// TwinCAT 3 PLC project MotorRuntime
// ProgramVersion: 3.1.4026.24
// libraries:
//   Tc2_Standard, * (Beckhoff Automation GmbH)
//   Tc2_System, * (Beckhoff Automation GmbH)
//   Tc3_Module, * (Beckhoff Automation GmbH)
// project tree:
//   DUTs/ DUT_AllocationSample.TcDUT, DUT_AxisCalibration.TcDUT, DUT_CommutationOverride.TcDUT, DUT_MotorDriverCommand.TcDUT, DUT_MotorDriverStatus.TcDUT, DUT_MotorFeedbackSnapshot.TcDUT
//   GVLs/ GVL_AllocationTransfer.TcGVL, GVL_MotorRuntime.TcGVL, GVL_MotorRuntimeInternal.TcGVL
//   POUs/ FB_AllocationTransfer.TcPOU, F_ArchRadToCstcaAngle.TcPOU, F_ArchWrap2Pi.TcPOU, FB_MotorCommandArbiter.TcPOU, FB_MotorIoWatchdog.TcPOU, FB_MotorRuntimeKernel.TcPOU, PRG_MotorRuntime.TcPOU
//   / PlcTask.TcTTO
// (motion and I/O tree: see PLC project experimentsequencer)
// real-time tasks:
//   TASK PlcTask1: cycle T#250us, priority 21, ADS port 351
//   TASK PlcTask: cycle T#125us, priority 20, ADS port 350
//   TASK StateTask: cycle T#10ms, priority 1, ADS port 352
// variable links:
//   ExperimentSequencer/ExperimentSequencer Instance <-> MotorRuntime/MotorRuntime Instance
//     PlcTask Inputs/GVL_ExperimentSequencer.motorFeedback <-> PlcTask Outputs/GVL_MotorRuntimeInternal.Feedback
//     PlcTask Outputs/GVL_ExperimentSequencer.commutationOverride <-> PlcTask Inputs/GVL_MotorRuntimeInternal.CommutationOverride
//     PlcTask Outputs/GVL_ExperimentSequencer.driveCommand <-> PlcTask Inputs/GVL_MotorRuntimeInternal.CommissioningCommand
//   MotorRuntime/MotorRuntime Instance <-> Device 3 (EtherCAT)/Drive 7 (XE2)
//     PlcTask Inputs/PRG_MotorRuntime.copleyActualCurrentCountModule1 <-> Module 1 (Cyclic torque with commutation angle Mode)/Cyclic torque with commutation angle Inputs/Torque actual value
//     PlcTask Inputs/PRG_MotorRuntime.copleyActualCurrentCountModule2 <-> Module 2 (Cyclic torque with commutation angle Mode)/Cyclic torque with commutation angle Inputs/Torque actual value
//     PlcTask Inputs/PRG_MotorRuntime.copleyInputToggle <-> WcState/InputToggle
//     PlcTask Inputs/PRG_MotorRuntime.copleyStatusWordModule1 <-> Module 1 (Cyclic torque with commutation angle Mode)/Cyclic torque with commutation angle Inputs/Status word
//     PlcTask Inputs/PRG_MotorRuntime.copleyStatusWordModule2 <-> Module 2 (Cyclic torque with commutation angle Mode)/Cyclic torque with commutation angle Inputs/Status word
//     PlcTask Inputs/PRG_MotorRuntime.copleyWcState <-> WcState/WcState
//     PlcTask Outputs/PRG_MotorRuntime.copleyCommutationAngleModule1 <-> Module 1 (Cyclic torque with commutation angle Mode)/Cyclic torque with commutation angle Outputs/Commutation angle
//     PlcTask Outputs/PRG_MotorRuntime.copleyCommutationAngleModule2 <-> Module 2 (Cyclic torque with commutation angle Mode)/Cyclic torque with commutation angle Outputs/Commutation angle
//     PlcTask Outputs/PRG_MotorRuntime.copleyControlWordModule1 <-> Module 1 (Cyclic torque with commutation angle Mode)/Cyclic torque with commutation angle Outputs/Control word
//     PlcTask Outputs/PRG_MotorRuntime.copleyControlWordModule2 <-> Module 2 (Cyclic torque with commutation angle Mode)/Cyclic torque with commutation angle Outputs/Control word
//     PlcTask Outputs/PRG_MotorRuntime.copleyTargetTorqueModule1 <-> Module 1 (Cyclic torque with commutation angle Mode)/Cyclic torque with commutation angle Outputs/Target Torque
//     PlcTask Outputs/PRG_MotorRuntime.copleyTargetTorqueModule2 <-> Module 2 (Cyclic torque with commutation angle Mode)/Cyclic torque with commutation angle Outputs/Target Torque
//   MotorRuntime/MotorRuntime Instance <-> Device 3 (EtherCAT)/Drive 8 (XE2)
//     PlcTask Inputs/PRG_MotorRuntime.copleyActualCurrentCountModule3 <-> Module 1 (Cyclic torque with commutation angle Mode)/Cyclic torque with commutation angle Inputs/Torque actual value
//     PlcTask Inputs/PRG_MotorRuntime.copleyActualCurrentCountModule4 <-> Module 2 (Cyclic torque with commutation angle Mode)/Cyclic torque with commutation angle Inputs/Torque actual value
//     PlcTask Inputs/PRG_MotorRuntime.copleyInputToggleDrive2 <-> WcState/InputToggle
//     PlcTask Inputs/PRG_MotorRuntime.copleyStatusWordModule3 <-> Module 1 (Cyclic torque with commutation angle Mode)/Cyclic torque with commutation angle Inputs/Status word
//     PlcTask Inputs/PRG_MotorRuntime.copleyStatusWordModule4 <-> Module 2 (Cyclic torque with commutation angle Mode)/Cyclic torque with commutation angle Inputs/Status word
//     PlcTask Inputs/PRG_MotorRuntime.copleyWcStateDrive2 <-> WcState/WcState
//     PlcTask Outputs/PRG_MotorRuntime.copleyCommutationAngleModule3 <-> Module 1 (Cyclic torque with commutation angle Mode)/Cyclic torque with commutation angle Outputs/Commutation angle
//     PlcTask Outputs/PRG_MotorRuntime.copleyCommutationAngleModule4 <-> Module 2 (Cyclic torque with commutation angle Mode)/Cyclic torque with commutation angle Outputs/Commutation angle
//     PlcTask Outputs/PRG_MotorRuntime.copleyControlWordModule3 <-> Module 1 (Cyclic torque with commutation angle Mode)/Cyclic torque with commutation angle Outputs/Control word
//     PlcTask Outputs/PRG_MotorRuntime.copleyControlWordModule4 <-> Module 2 (Cyclic torque with commutation angle Mode)/Cyclic torque with commutation angle Outputs/Control word
//     PlcTask Outputs/PRG_MotorRuntime.copleyTargetTorqueModule3 <-> Module 1 (Cyclic torque with commutation angle Mode)/Cyclic torque with commutation angle Outputs/Target Torque
//     PlcTask Outputs/PRG_MotorRuntime.copleyTargetTorqueModule4 <-> Module 2 (Cyclic torque with commutation angle Mode)/Cyclic torque with commutation angle Outputs/Target Torque
//   MotorRuntime/MotorRuntime Instance <-> Device 3 (EtherCAT)/Term 1 (EK1100)/Term 2 (EL5042)
//     PlcTask Inputs/PRG_MotorRuntime.encoderError <-> FB Inputs Channel 1/Status/Error
//     PlcTask Inputs/PRG_MotorRuntime.encoderInputToggle <-> WcState/InputToggle
//     PlcTask Inputs/PRG_MotorRuntime.encoderPositionRaw <-> FB Inputs Channel 1/Position
//     PlcTask Inputs/PRG_MotorRuntime.encoderReady <-> FB Inputs Channel 1/Status/Ready
//     PlcTask Inputs/PRG_MotorRuntime.encoderTxPdoState <-> FB Inputs Channel 1/Status/TxPDO State
//     PlcTask Inputs/PRG_MotorRuntime.encoderWcState <-> WcState/WcState
//   MotorRuntime/MotorRuntime Instance <-> TcCOM Objects/Object1 (motor_config)
//     PlcTask Inputs/GVL_MotorRuntime.Command/ControlWord <-> motor_config_Y/controlWord
//     PlcTask Outputs/GVL_MotorRuntime.Status/StatusWord <-> motor_config_U/statusWord
//   MotorRuntime/MotorRuntime Instance <-> TcCOM Objects/Object3 (linear_exp_2025a)
//     PlcTask Inputs/GVL_MotorRuntime.Command/TargetTorque <-> TcModuleOutput/LinearSystem/TargetTorque
//     PlcTask Outputs/GVL_MotorRuntime.Status/PositionActualValue <-> TcModuleInput/LinearSystem/Positionactualvalue
//     PlcTask Outputs/GVL_MotorRuntime.Status/TorqueActualValue <-> TcModuleInput/LinearSystem/Torqueactualvalue1
//     PlcTask Outputs/GVL_MotorRuntime.Status/VelocityActualValue <-> TcModuleInput/LinearSystem/Velocityactualvalue
//   MotorRuntime/MotorRuntime Instance <-> TcCOM Objects/Object3 (linear_exp_tunable_2025a)
//     PlcTask Inputs/GVL_MotorRuntime.Command/TargetTorque <-> TcModuleOutput/linearsystem/TargetTorque
//     PlcTask Outputs/GVL_MotorRuntime.Status/PositionActualValue <-> TcModuleInput/linearsystem/PositionActualValue
//     PlcTask Outputs/GVL_MotorRuntime.Status/TorqueActualValue <-> TcModuleInput/linearsystem/TorqueActualValue
//     PlcTask Outputs/GVL_MotorRuntime.Status/VelocityActualValue <-> TcModuleInput/linearsystem/VelocityActualValue

CONFIGURATION MotorRuntime
    RESOURCE PLC ON TwinCAT3
        TASK PlcTask(INTERVAL := T#250us, PRIORITY := 21);
        PROGRAM PRG_MotorRuntime WITH PlcTask : PRG_MotorRuntime;
    END_RESOURCE
END_CONFIGURATION

// ---- DUTs/DUT_AllocationSample.TcDUT
TYPE DUT_AllocationSample : STRUCT
    cycleIndex : UDINT;
    positionCount : DINT;
    velocityCount : DINT;
    virtualTorque : DINT;
    targetCurrent : ARRAY [1..4] OF DINT;
    actualCurrent : ARRAY [1..4] OF DINT;
    statusWord : ARRAY [1..4] OF DINT;
    faultId : UDINT;
    ioReady : DINT;
    period100ns : UDINT;
    requestId : UDINT;
END_STRUCT
END_TYPE

// ---- DUTs/DUT_AxisCalibration.TcDUT
TYPE DUT_AxisCalibration : STRUCT
    reference_position_count      : DINT;
    reference_commutation_angle   : UINT;
    electrical_direction          : INT;
END_STRUCT
END_TYPE

// ---- DUTs/DUT_CommutationOverride.TcDUT
TYPE DUT_CommutationOverride : STRUCT
    enable                 : BOOL;
    angle_offset_rad       : LREAL;
    axis_index             : UINT;
END_STRUCT
END_TYPE

// ---- DUTs/DUT_MotorDriverCommand.TcDUT
TYPE DUT_MotorDriverCommand : STRUCT
    ControlWord  : WORD;
    TargetTorque : INT;
END_STRUCT
END_TYPE

// ---- DUTs/DUT_MotorDriverStatus.TcDUT
TYPE DUT_MotorDriverStatus : STRUCT
    StatusWord          : WORD;
    PositionActualValue : DINT;
    VelocityActualValue : DINT;
    TorqueActualValue   : INT;
END_STRUCT
END_TYPE

// ---- DUTs/DUT_MotorFeedbackSnapshot.TcDUT
TYPE DUT_MotorFeedbackSnapshot : STRUCT
    encoder_position_raw       : DINT;
    encoder_velocity_raw       : DINT;
    copley_statusword          : WORD;
    copley_actual_current_count: INT;
    output_torque_count        : INT;
    fault_id                   : UDINT;
END_STRUCT
END_TYPE

// ---- GVLs/GVL_AllocationTransfer.TcGVL
{attribute 'qualified_only'}
VAR_GLOBAL CONSTANT
    SCHEMA_VERSION : UDINT := 2;
    SAMPLE_BYTES : UDINT := 80;
END_VAR
VAR_GLOBAL
    // Write parameters first, RequestId last. They are latched only at idle.
    RequestId : UDINT;
    RequestedEnabled : BOOL;
    RequestedPair : UINT := 1;
    RequestedBeta : LREAL;
    RequestedRatio : LREAL := 1.0;
    AckId : UDINT;
    RejectId : UDINT;
    Active : BOOL;
    Started : BOOL;
    Complete : BOOL;
    Pair : UINT;
    Beta : LREAL;
    Ratio : LREAL;
    Weights : ARRAY [1..2] OF LREAL := [1.0,1.0];
    FaultId : UDINT;
    // One coherent cycle is recorded by the common Simulink File Writer.
    Snapshot AT %Q* : DUT_AllocationSample;
END_VAR

// ---- GVLs/GVL_MotorRuntime.TcGVL
{attribute 'qualified_only'}
VAR_GLOBAL
    // The complete public virtual-CST boundary.
    Command AT %I* : DUT_MotorDriverCommand;
    Status  AT %Q* : DUT_MotorDriverStatus;
END_VAR

// ---- GVLs/GVL_MotorRuntimeInternal.TcGVL
{attribute 'qualified_only'}
VAR_GLOBAL CONSTANT
    AXIS_COUNT                    : UINT := 4;
    // Compile-time normal-CST topology: FALSE drives axes 1+2; TRUE drives axes 1..4.
    NORMAL_FOUR_AXIS_ENABLED      : BOOL := TRUE;
    COUNTS_PER_ELECTRICAL_PERIOD : DINT := 360000;
    // Public virtual CST follows CiA 402 rated torque / 1000. The physical
    // Copley channels retain their high-resolution 0.1 A / 1000 scaling.
    VIRTUAL_RATED_TORQUE_EQUIVALENT_CURRENT_MA : DINT := 2000;
    COPLEY_INTERNAL_CURRENT_MA_PER_1000_COUNT   : DINT := 100;
    // Inclusive raw Panasonic encoder windows. Adjacent windows overlap over
    // the measured Core1~2, Core2~3, and Core3~4 transition regions.
    TORQUE_LINKAGE_LOWER_COUNT : ARRAY [1..AXIS_COUNT] OF DINT := [
        54054804, 55809159, 59369714, 63068811];
    TORQUE_LINKAGE_UPPER_COUNT : ARRAY [1..AXIS_COUNT] OF DINT := [
        57600015, 61230980, 64809681, 66655810];
    // Each boundary may vary by 10% of the largest measured segment width:
    // ceil((61230980 - 59369714) * 0.10). Extend both ends for either direction.
    TORQUE_LINKAGE_MARGIN_COUNT : DINT := 186127;
END_VAR

VAR_GLOBAL RETAIN
    // Registered values for all four axes mirror the checked-in authoritative
    // manifest. Set validity false before replacing any complete record.
    RegisteredReferenceValid : ARRAY [1..AXIS_COUNT] OF BOOL := [TRUE, TRUE, TRUE, TRUE];
    RegisteredReference : ARRAY [1..AXIS_COUNT] OF DUT_AxisCalibration := [
        (reference_position_count := 54984708,
         reference_commutation_angle := 49480,
         electrical_direction := 1),
        (reference_position_count := 58408617,
         reference_commutation_angle := 17933,
         electrical_direction := 1),
        (reference_position_count := 61902867,
         reference_commutation_angle := 63448,
         electrical_direction := 1),
        (reference_position_count := 65824016,
         reference_commutation_angle := 57717,
         electrical_direction := 1)
    ];
END_VAR

VAR_GLOBAL
    // Commissioning writes provisional/interim references here. Normal CST
    // never reads this non-retained array.
    CommissioningReference : ARRAY [1..AXIS_COUNT] OF DUT_AxisCalibration;

    // These linked process-image symbols are private commissioning channels.
    // They are deliberately excluded from GVL_MotorRuntime.
    CommissioningCommand AT %I* : DUT_MotorDriverCommand;
    CommutationOverride  AT %I* : DUT_CommutationOverride;

    // One-shot operator acknowledgement for a latched I/O-watchdog fault.
    // PRG_MotorRuntime clears this after sampling it. A reset is accepted only
    // while the selected command is explicitly zero and both slaves are healthy.
    IoWatchdogResetRequest : BOOL;

    // Private commissioning feedback.
    Feedback AT %Q* : DUT_MotorFeedbackSnapshot;
END_VAR

// ---- POUs/PRG_MotorRuntime.TcPOU
PROGRAM PRG_MotorRuntime
VAR
    fbMotor : FB_MotorRuntimeKernel;
    fbArbiter : FB_MotorCommandArbiter;
    fbIoWatchdog : FB_MotorIoWatchdog;
    fbAllocation : FB_AllocationTransfer;

    AllocationRequestId AT %I* : UDINT;

    encoderPositionRaw        AT %I* : ULINT;
    encoderReady              AT %I* : BOOL;
    encoderError              AT %I* : BOOL;
    encoderTxPdoState         AT %I* : BOOL;
    encoderWcState            AT %I* : BOOL;
    encoderInputToggle        AT %I* : BOOL;
    copleyWcState             AT %I* : BOOL;
    copleyInputToggle         AT %I* : BOOL;
    copleyWcStateDrive2       AT %I* : BOOL;
    copleyInputToggleDrive2   AT %I* : BOOL;
    copleyStatusWordModule1         AT %I* : WORD;
    copleyActualCurrentCountModule1 AT %I* : INT;
    copleyStatusWordModule2         AT %I* : WORD;
    copleyActualCurrentCountModule2 AT %I* : INT;
    copleyStatusWordModule3         AT %I* : WORD;
    copleyActualCurrentCountModule3 AT %I* : INT;
    copleyStatusWordModule4         AT %I* : WORD;
    copleyActualCurrentCountModule4 AT %I* : INT;

    copleyControlWordModule1      AT %Q* : WORD;
    copleyTargetTorqueModule1     AT %Q* : INT;
    copleyCommutationAngleModule1 AT %Q* : UINT;
    copleyControlWordModule2      AT %Q* : WORD;
    copleyTargetTorqueModule2     AT %Q* : INT;
    copleyCommutationAngleModule2 AT %Q* : UINT;
    copleyControlWordModule3      AT %Q* : WORD;
    copleyTargetTorqueModule3     AT %Q* : INT;
    copleyCommutationAngleModule3 AT %Q* : UINT;
    copleyControlWordModule4      AT %Q* : WORD;
    copleyTargetTorqueModule4     AT %Q* : INT;
    copleyCommutationAngleModule4 AT %Q* : UINT;

    copleyStatusWord         : ARRAY [1..GVL_MotorRuntimeInternal.AXIS_COUNT] OF WORD;
    copleyActualCurrentCount : ARRAY [1..GVL_MotorRuntimeInternal.AXIS_COUNT] OF INT;
    encoderPositionActualRaw : DINT;
    encoderVelocityActualRaw : DINT;
    previousEncoderPositionRaw : DINT;
    encoderPositionInitialized : BOOL;
    taskIndex                  : DINT;
    cycleTime100ns             : UDINT;
    taskPeriod_s               : LREAL := 0.00025;
END_VAR

taskIndex := GETCURTASKINDEXEX();
IF taskIndex > 0 THEN
    cycleTime100ns := TwinCAT_SystemInfoVarList._TaskInfo[taskIndex].CycleTime;
    IF cycleTime100ns > 0 THEN
        taskPeriod_s := UDINT_TO_LREAL(cycleTime100ns) * 1.0E-7;
    END_IF
END_IF

encoderPositionActualRaw := ULINT_TO_DINT(encoderPositionRaw);
IF encoderPositionInitialized THEN
    // Position is 0.1 um/count; velocity is published in 1 um/s/count.
    encoderVelocityActualRaw := LREAL_TO_DINT(
        DINT_TO_LREAL(encoderPositionActualRaw - previousEncoderPositionRaw)
        * 0.1 / taskPeriod_s);
ELSE
    encoderVelocityActualRaw := 0;
    encoderPositionInitialized := TRUE;
END_IF
previousEncoderPositionRaw := encoderPositionActualRaw;

copleyStatusWord[1] := copleyStatusWordModule1;
copleyActualCurrentCount[1] := copleyActualCurrentCountModule1;
copleyStatusWord[2] := copleyStatusWordModule2;
copleyActualCurrentCount[2] := copleyActualCurrentCountModule2;
copleyStatusWord[3] := copleyStatusWordModule3;
copleyActualCurrentCount[3] := copleyActualCurrentCountModule3;
copleyStatusWord[4] := copleyStatusWordModule4;
copleyActualCurrentCount[4] := copleyActualCurrentCountModule4;

fbArbiter(
    NormalCommand := GVL_MotorRuntime.Command,
    CommissioningCommand := GVL_MotorRuntimeInternal.CommissioningCommand,
    CommutationOverride := GVL_MotorRuntimeInternal.CommutationOverride);

fbMotor(
    Command := fbArbiter.SelectedCommand,
    CommutationOverride := fbArbiter.SelectedCommutationOverride,
    RegisteredReferenceValid := GVL_MotorRuntimeInternal.RegisteredReferenceValid,
    RegisteredReference := GVL_MotorRuntimeInternal.RegisteredReference,
    CommissioningReference := GVL_MotorRuntimeInternal.CommissioningReference,
    EncoderPositionActualRaw := encoderPositionActualRaw,
    EncoderVelocityActualRaw := encoderVelocityActualRaw,
    CopleyStatusWord := copleyStatusWord,
    CopleyActualCurrentCount := copleyActualCurrentCount);

fbIoWatchdog(
    TaskPeriod_s := taskPeriod_s,
    EncoderWcState := encoderWcState,
    EncoderInputToggle := encoderInputToggle,
    EncoderReady := encoderReady,
    EncoderError := encoderError,
    EncoderTxPdoState := encoderTxPdoState,
    CopleyWcState := copleyWcState,
    CopleyInputToggle := copleyInputToggle,
    Copley2WcState := copleyWcStateDrive2,
    Copley2InputToggle := copleyInputToggleDrive2,
    ResetRequest :=
        GVL_MotorRuntimeInternal.IoWatchdogResetRequest
        AND (fbArbiter.CommissioningActive
             OR NOT fbArbiter.CommissioningActive),
    CommandIsZero :=
        (fbArbiter.SelectedCommand.ControlWord = WORD#16#0000)
        AND (fbArbiter.SelectedCommand.TargetTorque = 0));
// Consume the operator acknowledgement as a one-cycle request. Keeping it
// separate from the command prevents automatic re-arm after communication
// recovers while an idle 0/0 command happens to be present.
GVL_MotorRuntimeInternal.IoWatchdogResetRequest := FALSE;

fbAllocation(
    Command := fbArbiter.SelectedCommand,
    RuntimeRequestId := AllocationRequestId,
    CommissioningActive := fbArbiter.CommissioningActive,
    SourceControl := fbMotor.CopleyControlWord,
    SourceTorque := fbMotor.CopleyTargetTorque,
    StatusWord := copleyStatusWord,
    ActualCurrent := copleyActualCurrentCount,
    PositionCount := encoderPositionActualRaw,
    VelocityCount := encoderVelocityActualRaw,
    IoReady := fbIoWatchdog.SafeToDrive,
    SourceFaultId := fbMotor.FaultId,
    Period100ns := cycleTime100ns);

GVL_MotorRuntime.Status := fbMotor.Status;
GVL_MotorRuntimeInternal.Feedback := fbMotor.Feedback;
IF GVL_AllocationTransfer.FaultId <> 0 THEN
    GVL_MotorRuntimeInternal.Feedback.fault_id := GVL_AllocationTransfer.FaultId;
END_IF
IF (fbArbiter.CommissioningActive OR NOT fbArbiter.CommissioningActive)
   AND fbIoWatchdog.Fault THEN
    GVL_MotorRuntimeInternal.Feedback.fault_id := fbIoWatchdog.FaultId;
END_IF

IF (fbArbiter.CommissioningActive OR NOT fbArbiter.CommissioningActive)
   AND fbIoWatchdog.SafeToDrive THEN
    copleyControlWordModule1 := fbAllocation.Control[1];
    copleyTargetTorqueModule1 := fbAllocation.Torque[1];
    copleyCommutationAngleModule1 := fbMotor.CopleyCommutationAngle[1];
    copleyControlWordModule2 := fbAllocation.Control[2];
    copleyTargetTorqueModule2 := fbAllocation.Torque[2];
    copleyCommutationAngleModule2 := fbMotor.CopleyCommutationAngle[2];
    copleyControlWordModule3 := fbAllocation.Control[3];
    copleyTargetTorqueModule3 := fbAllocation.Torque[3];
    copleyCommutationAngleModule3 := fbMotor.CopleyCommutationAngle[3];
    copleyControlWordModule4 := fbAllocation.Control[4];
    copleyTargetTorqueModule4 := fbAllocation.Torque[4];
    copleyCommutationAngleModule4 := fbMotor.CopleyCommutationAngle[4];
ELSE
    // This is the final gate before the physical PDO outputs. It remains
    // effective even if the TcCOM controller continues to request torque.
    copleyControlWordModule1 := WORD#16#0000;
    copleyTargetTorqueModule1 := 0;
    copleyCommutationAngleModule1 := 0;
    copleyControlWordModule2 := WORD#16#0000;
    copleyTargetTorqueModule2 := 0;
    copleyCommutationAngleModule2 := 0;
    copleyControlWordModule3 := WORD#16#0000;
    copleyTargetTorqueModule3 := 0;
    copleyCommutationAngleModule3 := 0;
    copleyControlWordModule4 := WORD#16#0000;
    copleyTargetTorqueModule4 := 0;
    copleyCommutationAngleModule4 := 0;
END_IF

END_PROGRAM

// ---- POUs/FB_MotorRuntimeKernel.TcPOU
FUNCTION_BLOCK FB_MotorRuntimeKernel
VAR_INPUT
    Command                    : DUT_MotorDriverCommand;
    CommutationOverride        : DUT_CommutationOverride;
    RegisteredReferenceValid   : ARRAY [1..GVL_MotorRuntimeInternal.AXIS_COUNT] OF BOOL;
    RegisteredReference        : ARRAY [1..GVL_MotorRuntimeInternal.AXIS_COUNT] OF DUT_AxisCalibration;
    CommissioningReference     : ARRAY [1..GVL_MotorRuntimeInternal.AXIS_COUNT] OF DUT_AxisCalibration;
    EncoderPositionActualRaw : DINT;
    EncoderVelocityActualRaw : DINT;
    CopleyStatusWord           : ARRAY [1..GVL_MotorRuntimeInternal.AXIS_COUNT] OF WORD;
    CopleyActualCurrentCount   : ARRAY [1..GVL_MotorRuntimeInternal.AXIS_COUNT] OF INT;
END_VAR
VAR_OUTPUT
    Status                     : DUT_MotorDriverStatus;
    Feedback                   : DUT_MotorFeedbackSnapshot;
    CopleyControlWord          : ARRAY [1..GVL_MotorRuntimeInternal.AXIS_COUNT] OF WORD;
    CopleyTargetTorque         : ARRAY [1..GVL_MotorRuntimeInternal.AXIS_COUNT] OF INT;
    CopleyCommutationAngle     : ARRAY [1..GVL_MotorRuntimeInternal.AXIS_COUNT] OF UINT;
    Fault                      : BOOL;
    FaultId                    : UDINT;
END_VAR
VAR
    Ready                      : BOOL;
    limitedCommand             : DUT_MotorDriverCommand;
    i                          : INT;
    axisIndex                  : UINT;
    axisIndexInt               : INT;
    axisBit                    : WORD;
    overrideAxisValid          : BOOL;
    copleyFaultByAxis          : ARRAY [1..GVL_MotorRuntimeInternal.AXIS_COUNT] OF BOOL;
    copleyFault                : BOOL;
    overrideRequired           : BOOL;
    positionDeltaCount         : LREAL;
    referenceAngleRad          : LREAL;
    thetaCmd                   : LREAL;
    aggregateMask              : WORD;
    aggregateActualDint        : DINT;
    aggregateOutputDint        : DINT;
    aggregateActual            : INT;
    aggregateOutput            : INT;
    statusActualDint           : DINT;
    statusActualNumerator      : DINT;
    statusActualDenominator    : DINT;
    statusActual               : INT;
    scaledTorqueDint           : DINT;
    statusWordAggregate        : WORD;
    feedbackStatusWord         : WORD;
    statusStateBits            : WORD;
    axisStateMasked            : WORD;
    minimumStateRank           : INT;
    axisStateRank              : INT;
    anyFaultReactionActive     : BOOL;
    anyFaultState              : BOOL;
    anyQuickStopActive         : BOOL;
    registeredReferencesValid  : BOOL;
    normalAxisActive           : ARRAY [1..GVL_MotorRuntimeInternal.AXIS_COUNT] OF BOOL;
    torqueAxisLinked           : ARRAY [1..GVL_MotorRuntimeInternal.AXIS_COUNT] OF BOOL;
    activeAxisCount            : DINT;
END_VAR

axisIndex := 1;
overrideAxisValid := TRUE;
copleyFault := FALSE;
minimumStateRank := 32767;
anyFaultReactionActive := FALSE;
anyFaultState := FALSE;
anyQuickStopActive := FALSE;
registeredReferencesValid := TRUE;
activeAxisCount := 0;

IF CommutationOverride.enable THEN
    IF (CommutationOverride.axis_index < 1) OR (CommutationOverride.axis_index > GVL_MotorRuntimeInternal.AXIS_COUNT) THEN
        overrideAxisValid := FALSE;
    ELSE
        axisIndex := CommutationOverride.axis_index;
    END_IF
END_IF

overrideRequired := CommutationOverride.enable;
axisIndexInt := UINT_TO_INT(axisIndex);

limitedCommand := Command;
// Private commissioning commands already use the physical 0.1 A / 1000
// representation. Convert only the public virtual-CST rated-torque command.
IF NOT overrideRequired THEN
    scaledTorqueDint :=
        INT_TO_DINT(Command.TargetTorque)
        * GVL_MotorRuntimeInternal.VIRTUAL_RATED_TORQUE_EQUIVALENT_CURRENT_MA
        / GVL_MotorRuntimeInternal.COPLEY_INTERNAL_CURRENT_MA_PER_1000_COUNT;
    IF scaledTorqueDint > 32767 THEN
        limitedCommand.TargetTorque := DINT_TO_INT(32767);
    ELSIF scaledTorqueDint < -32768 THEN
        limitedCommand.TargetTorque := DINT_TO_INT(-32768);
    ELSE
        limitedCommand.TargetTorque := DINT_TO_INT(scaledTorqueDint);
    END_IF
END_IF

FOR i := 1 TO UINT_TO_INT(GVL_MotorRuntimeInternal.AXIS_COUNT) DO
    normalAxisActive[i] :=
        (i <= 2)
        OR GVL_MotorRuntimeInternal.NORMAL_FOUR_AXIS_ENABLED;
    torqueAxisLinked[i] :=
        normalAxisActive[i]
        AND (EncoderPositionActualRaw >= GVL_MotorRuntimeInternal.TORQUE_LINKAGE_LOWER_COUNT[i]
            - GVL_MotorRuntimeInternal.TORQUE_LINKAGE_MARGIN_COUNT)
        AND (EncoderPositionActualRaw <= GVL_MotorRuntimeInternal.TORQUE_LINKAGE_UPPER_COUNT[i]
            + GVL_MotorRuntimeInternal.TORQUE_LINKAGE_MARGIN_COUNT);
    CopleyControlWord[i] := WORD#16#0000;
    CopleyTargetTorque[i] := 0;
    CopleyCommutationAngle[i] := 0;

    copleyFaultByAxis[i] :=
        (CopleyStatusWord[i] AND WORD#16#0008) <> WORD#16#0000;
    IF normalAxisActive[i] THEN
        activeAxisCount := activeAxisCount + 1;
        registeredReferencesValid :=
            registeredReferencesValid AND RegisteredReferenceValid[i];
        axisStateMasked := CopleyStatusWord[i] AND WORD#16#006F;
        IF (CopleyStatusWord[i] AND WORD#16#004F) = WORD#16#000F THEN
            anyFaultReactionActive := TRUE;
            axisStateRank := 0;
        ELSIF (CopleyStatusWord[i] AND WORD#16#004F) = WORD#16#0008 THEN
            anyFaultState := TRUE;
            axisStateRank := 0;
        ELSIF axisStateMasked = WORD#16#0007 THEN
            anyQuickStopActive := TRUE;
            axisStateRank := 0;
        ELSIF (CopleyStatusWord[i] AND WORD#16#004F) = WORD#16#0040 THEN
            axisStateRank := 1;
        ELSIF axisStateMasked = WORD#16#0021 THEN
            axisStateRank := 2;
        ELSIF axisStateMasked = WORD#16#0023 THEN
            axisStateRank := 3;
        ELSIF axisStateMasked = WORD#16#0027 THEN
            axisStateRank := 4;
        ELSE
            axisStateRank := 0;
        END_IF
        IF axisStateRank < minimumStateRank THEN
            minimumStateRank := axisStateRank;
        END_IF
    END_IF
END_FOR

copleyFault := FALSE;
IF overrideRequired AND overrideAxisValid THEN
    copleyFault := copleyFaultByAxis[axisIndexInt];
ELSE
    FOR i := 1 TO UINT_TO_INT(GVL_MotorRuntimeInternal.AXIS_COUNT) DO
        IF normalAxisActive[i] THEN
            copleyFault := copleyFault OR copleyFaultByAxis[i];
        END_IF
    END_FOR
END_IF

IF overrideRequired THEN
    Ready :=
        NOT copleyFault
        AND overrideAxisValid;
ELSE
    Ready := registeredReferencesValid;
END_IF
Fault := FALSE;
FaultId := 0;

IF NOT overrideAxisValid THEN
    Fault := TRUE;
    FaultId := 611; // invalid commutation override axis
ELSIF copleyFault THEN
    Fault := TRUE;
    FaultId := 506; // physical drive fault
ELSIF NOT overrideRequired
      AND NOT registeredReferencesValid
      AND ((Command.ControlWord <> WORD#16#0000)
           OR (Command.TargetTorque <> 0)) THEN
    Fault := TRUE;
    FaultId := 612; // normal reference not registered for every active axis
END_IF

FOR i := 1 TO UINT_TO_INT(GVL_MotorRuntimeInternal.AXIS_COUNT) DO
    IF overrideRequired AND overrideAxisValid AND (i = axisIndexInt) THEN
        // Commissioning is deliberately isolated from the retained normal-CST
        // references and only drives its explicitly selected physical axis.
        // Convert before subtraction so the full DINT endpoint delta is safe.
        positionDeltaCount :=
            DINT_TO_LREAL(EncoderPositionActualRaw)
            - DINT_TO_LREAL(
                CommissioningReference[i].reference_position_count);
        referenceAngleRad :=
            UINT_TO_LREAL(
                CommissioningReference[i].reference_commutation_angle)
            * 6.2831853071795864769 / 65536.0;

        thetaCmd := F_ArchWrap2Pi(
            referenceAngleRad
            + INT_TO_LREAL(CommissioningReference[i].electrical_direction)
              * 6.2831853071795864769 * positionDeltaCount
              / DINT_TO_LREAL(GVL_MotorRuntimeInternal.COUNTS_PER_ELECTRICAL_PERIOD)
            + CommutationOverride.angle_offset_rad);
        CopleyCommutationAngle[i] := F_ArchRadToCstcaAngle(thetaCmd);
    ELSIF NOT overrideRequired AND Ready AND normalAxisActive[i] THEN
        // Normal CST starts only after every active axis record was registered
        // and read back. Each active axis still uses only its own record.
        positionDeltaCount :=
            DINT_TO_LREAL(EncoderPositionActualRaw)
            - DINT_TO_LREAL(RegisteredReference[i].reference_position_count);
        referenceAngleRad :=
            UINT_TO_LREAL(RegisteredReference[i].reference_commutation_angle)
            * 6.2831853071795864769 / 65536.0;
        thetaCmd := F_ArchWrap2Pi(
            referenceAngleRad
            + INT_TO_LREAL(RegisteredReference[i].electrical_direction)
              * 6.2831853071795864769 * positionDeltaCount
              / DINT_TO_LREAL(GVL_MotorRuntimeInternal.COUNTS_PER_ELECTRICAL_PERIOD));
        CopleyCommutationAngle[i] := F_ArchRadToCstcaAngle(thetaCmd);
    END_IF
END_FOR

IF overrideRequired THEN
    IF Ready THEN
        CopleyControlWord[axisIndexInt] := limitedCommand.ControlWord;
        CopleyTargetTorque[axisIndexInt] := limitedCommand.TargetTorque;
    END_IF
ELSIF Ready THEN
    // Keep every configured drive enabled and commutated, but apply torque only
    // while its motor core is linked to the shared mover. Overlapping windows
    // keep both neighboring cores active through each measured transition.
    FOR i := 1 TO UINT_TO_INT(GVL_MotorRuntimeInternal.AXIS_COUNT) DO
        IF normalAxisActive[i] THEN
            CopleyControlWord[i] := limitedCommand.ControlWord;
            IF torqueAxisLinked[i] THEN
                CopleyTargetTorque[i] := limitedCommand.TargetTorque;
            END_IF
        END_IF
    END_FOR
END_IF

aggregateMask := WORD#16#0000;
IF overrideRequired AND overrideAxisValid THEN
    aggregateMask := SHL(WORD#16#0001, axisIndexInt - 1);
ELSE
    FOR i := 1 TO UINT_TO_INT(GVL_MotorRuntimeInternal.AXIS_COUNT) DO
        IF normalAxisActive[i] THEN
            aggregateMask := aggregateMask OR SHL(WORD#16#0001, i - 1);
        END_IF
    END_FOR
END_IF

aggregateActualDint := 0;
aggregateOutputDint := 0;
statusActualDint := 0;
FOR i := 1 TO UINT_TO_INT(GVL_MotorRuntimeInternal.AXIS_COUNT) DO
    IF normalAxisActive[i] THEN
        statusActualDint :=
            statusActualDint + INT_TO_DINT(CopleyActualCurrentCount[i]);
    END_IF
    axisBit := SHL(WORD#16#0001, i - 1);
    IF (aggregateMask AND axisBit) <> WORD#16#0000 THEN
        aggregateActualDint := aggregateActualDint + INT_TO_DINT(CopleyActualCurrentCount[i]);
        aggregateOutputDint := aggregateOutputDint + INT_TO_DINT(CopleyTargetTorque[i]);
    END_IF
END_FOR

// The public virtual drive represents the configured active axes, not their
// sum. Convert their average physical current count back to rated torque / 1000,
// with symmetric rounding around zero.
statusActualNumerator :=
    statusActualDint
    * GVL_MotorRuntimeInternal.COPLEY_INTERNAL_CURRENT_MA_PER_1000_COUNT;
statusActualDenominator :=
    activeAxisCount
    * GVL_MotorRuntimeInternal.VIRTUAL_RATED_TORQUE_EQUIVALENT_CURRENT_MA;
IF statusActualNumerator >= 0 THEN
    statusActualNumerator := statusActualNumerator + statusActualDenominator / 2;
ELSE
    statusActualNumerator := statusActualNumerator - statusActualDenominator / 2;
END_IF
statusActual := DINT_TO_INT(statusActualNumerator / statusActualDenominator);

IF aggregateActualDint > 32767 THEN
    aggregateActual := DINT_TO_INT(32767);
ELSIF aggregateActualDint < -32768 THEN
    aggregateActual := DINT_TO_INT(-32768);
ELSE
    aggregateActual := DINT_TO_INT(aggregateActualDint);
END_IF

IF aggregateOutputDint > 32767 THEN
    aggregateOutput := DINT_TO_INT(32767);
ELSIF aggregateOutputDint < -32768 THEN
    aggregateOutput := DINT_TO_INT(-32768);
ELSE
    aggregateOutput := DINT_TO_INT(aggregateOutputDint);
END_IF

// The public virtual drive reports one canonical CiA 402 state value. Copley
// auxiliary/manufacturer bits (for example 0x1600) remain available in the
// private per-axis diagnostics, but must not obscure the public state. A
// lagging or faulted active axis therefore remains visible without leaking
// drive-specific bits into the virtual-CST boundary. Inactive axes are private.
IF anyFaultReactionActive THEN
    statusStateBits := WORD#16#000F;
ELSIF anyFaultState THEN
    statusStateBits := WORD#16#0008;
ELSIF anyQuickStopActive THEN
    statusStateBits := WORD#16#0007;
ELSIF minimumStateRank >= 4 THEN
    statusStateBits := WORD#16#0027;
ELSIF minimumStateRank = 3 THEN
    statusStateBits := WORD#16#0023;
ELSIF minimumStateRank = 2 THEN
    statusStateBits := WORD#16#0021;
ELSIF minimumStateRank = 1 THEN
    statusStateBits := WORD#16#0040;
ELSE
    statusStateBits := WORD#16#0000;
END_IF
statusWordAggregate := statusStateBits;

// Private commissioning feedback remains scoped to its selected physical axis.
IF overrideRequired AND overrideAxisValid THEN
    feedbackStatusWord := CopleyStatusWord[axisIndexInt];
ELSE
    feedbackStatusWord := statusWordAggregate;
END_IF
// Public CiA 402 fault bit 3 reflects only a physical Copley fault aggregated
// above. Internal runtime safety faults stay private in Feedback/FaultId; they
// cannot be cleared by a drive reset and must not force MotorDriver to 0x0080.

Status.StatusWord := statusWordAggregate;
Status.PositionActualValue := EncoderPositionActualRaw;
Status.VelocityActualValue := EncoderVelocityActualRaw;
Status.TorqueActualValue := statusActual;

Feedback.encoder_position_raw := EncoderPositionActualRaw;
Feedback.encoder_velocity_raw := EncoderVelocityActualRaw;
Feedback.copley_statusword := feedbackStatusWord;
Feedback.copley_actual_current_count := aggregateActual;
Feedback.output_torque_count := aggregateOutput;
Feedback.fault_id := FaultId;

END_FUNCTION_BLOCK

// ---- POUs/F_ArchWrap2Pi.TcPOU
FUNCTION F_ArchWrap2Pi : LREAL
VAR_INPUT
    theta : LREAL;
END_VAR
VAR CONSTANT
    TWO_PI : LREAL := 6.2831853071795864769;
END_VAR
VAR
    y : LREAL;
END_VAR

y := theta - TWO_PI * LREAL_TO_DINT(theta / TWO_PI);
WHILE y < 0.0 DO
    y := y + TWO_PI;
END_WHILE
WHILE y >= TWO_PI DO
    y := y - TWO_PI;
END_WHILE
F_ArchWrap2Pi := y;

END_FUNCTION

// ---- POUs/F_ArchRadToCstcaAngle.TcPOU
FUNCTION F_ArchRadToCstcaAngle : UINT
VAR_INPUT
    theta : LREAL;
END_VAR
VAR CONSTANT
    TWO_PI : LREAL := 6.2831853071795864769;
END_VAR
VAR
    wrapped : LREAL;
    counts  : DINT;
END_VAR

wrapped := F_ArchWrap2Pi(theta);
counts := LREAL_TO_DINT(wrapped / TWO_PI * 65536.0);
IF counts >= 65536 THEN
    counts := counts - 65536;
ELSIF counts < 0 THEN
    counts := counts + 65536;
END_IF
F_ArchRadToCstcaAngle := DINT_TO_UINT(counts);

END_FUNCTION

// ---- POUs/FB_MotorCommandArbiter.TcPOU
FUNCTION_BLOCK FB_MotorCommandArbiter
VAR_INPUT
    NormalCommand         : DUT_MotorDriverCommand;
    CommissioningCommand  : DUT_MotorDriverCommand;
    CommutationOverride   : DUT_CommutationOverride;
END_VAR
VAR_OUTPUT
    SelectedCommand             : DUT_MotorDriverCommand;
    SelectedCommutationOverride : DUT_CommutationOverride;
    CommissioningActive         : BOOL;
END_VAR
VAR
    normalCommandZero      : BOOL;
    commissioningRequested : BOOL;
END_VAR

normalCommandZero :=
    (NormalCommand.ControlWord = WORD#16#0000)
    AND (NormalCommand.TargetTorque = 0);

// The public virtual-CST command is the normal runtime authority. Do not
// reinterpret, pulse-limit, range-filter, or insert zero cycles into its
// ControlWord/TargetTorque pair. The physical drive owns its safety limits.
// Commissioning can take ownership only while the normal interface is idle.
commissioningRequested :=
    CommutationOverride.enable AND normalCommandZero;

SelectedCommutationOverride.enable := FALSE;
SelectedCommutationOverride.angle_offset_rad :=
    CommutationOverride.angle_offset_rad;
SelectedCommutationOverride.axis_index := CommutationOverride.axis_index;

IF commissioningRequested THEN
    SelectedCommand.ControlWord := CommissioningCommand.ControlWord;
    SelectedCommand.TargetTorque := CommissioningCommand.TargetTorque;
    SelectedCommutationOverride.enable := TRUE;
    CommissioningActive := TRUE;
ELSE
    SelectedCommand.ControlWord := NormalCommand.ControlWord;
    SelectedCommand.TargetTorque := NormalCommand.TargetTorque;
    CommissioningActive := FALSE;
END_IF

END_FUNCTION_BLOCK

// ---- POUs/FB_MotorIoWatchdog.TcPOU
FUNCTION_BLOCK FB_MotorIoWatchdog
VAR_INPUT
    TaskPeriod_s       : LREAL := 0.00025;
    ToggleTimeout_s    : LREAL := 0.010;
    EncoderWcState     : BOOL;
    EncoderInputToggle : BOOL;
    EncoderReady       : BOOL;
    EncoderError       : BOOL;
    EncoderTxPdoState  : BOOL;
    CopleyWcState      : BOOL;
    CopleyInputToggle  : BOOL;
    Copley2WcState     : BOOL;
    Copley2InputToggle : BOOL;
    ResetRequest       : BOOL;
    CommandIsZero      : BOOL;
END_VAR
VAR_OUTPUT
    SafeToDrive                 : BOOL;
    Fault                       : BOOL;
    FaultId                     : UDINT;
END_VAR
VAR
    EncoderInputStaleCycles  : UDINT;
    CopleyInputStaleCycles   : UDINT;
    Copley2InputStaleCycles  : UDINT;
    lastEncoderInputToggle   : BOOL;
    lastCopleyInputToggle    : BOOL;
    lastCopley2InputToggle   : BOOL;
    encoderToggleSeen        : BOOL;
    copleyToggleSeen         : BOOL;
    copley2ToggleSeen        : BOOL;
    encoderToggleHealthy     : BOOL;
    copleyToggleHealthy      : BOOL;
    copley2ToggleHealthy     : BOOL;
END_VAR

IF EncoderInputToggle <> lastEncoderInputToggle THEN
    EncoderInputStaleCycles := 0;
    encoderToggleSeen := TRUE;
    lastEncoderInputToggle := EncoderInputToggle;
ELSIF EncoderInputStaleCycles < UDINT#16#FFFFFFFF THEN
    EncoderInputStaleCycles := EncoderInputStaleCycles + 1;
END_IF

IF CopleyInputToggle <> lastCopleyInputToggle THEN
    CopleyInputStaleCycles := 0;
    copleyToggleSeen := TRUE;
    lastCopleyInputToggle := CopleyInputToggle;
ELSIF CopleyInputStaleCycles < UDINT#16#FFFFFFFF THEN
    CopleyInputStaleCycles := CopleyInputStaleCycles + 1;
END_IF

IF Copley2InputToggle <> lastCopley2InputToggle THEN
    Copley2InputStaleCycles := 0;
    copley2ToggleSeen := TRUE;
    lastCopley2InputToggle := Copley2InputToggle;
ELSIF Copley2InputStaleCycles < UDINT#16#FFFFFFFF THEN
    Copley2InputStaleCycles := Copley2InputStaleCycles + 1;
END_IF

encoderToggleHealthy :=
    encoderToggleSeen
    AND (UDINT_TO_LREAL(EncoderInputStaleCycles) * TaskPeriod_s <= ToggleTimeout_s);
copleyToggleHealthy :=
    copleyToggleSeen
    AND (UDINT_TO_LREAL(CopleyInputStaleCycles) * TaskPeriod_s <= ToggleTimeout_s);
copley2ToggleHealthy :=
    copley2ToggleSeen
    AND (UDINT_TO_LREAL(Copley2InputStaleCycles) * TaskPeriod_s <= ToggleTimeout_s);

// The first fault is retained so post-mortem data identifies the initiating
// slave. Re-arming requires valid telegrams and an explicit zero command.
IF NOT Fault THEN
    IF EncoderWcState OR EncoderTxPdoState
       OR (encoderToggleSeen AND (EncoderError OR NOT EncoderReady)) THEN
        Fault := TRUE;
        FaultId := 620; // Encoder EtherCAT process data invalid
    ELSIF CopleyWcState OR Copley2WcState THEN
        Fault := TRUE;
        FaultId := 622; // Copley EtherCAT process data invalid
    ELSIF NOT encoderToggleHealthy
          AND (UDINT_TO_LREAL(EncoderInputStaleCycles) * TaskPeriod_s > ToggleTimeout_s) THEN
        Fault := TRUE;
        FaultId := 621; // Encoder valid input telegram stale
    ELSIF NOT copleyToggleHealthy
          AND (UDINT_TO_LREAL(CopleyInputStaleCycles) * TaskPeriod_s > ToggleTimeout_s) THEN
        Fault := TRUE;
        FaultId := 623; // Copley valid input telegram stale
    ELSIF NOT copley2ToggleHealthy
          AND (UDINT_TO_LREAL(Copley2InputStaleCycles) * TaskPeriod_s > ToggleTimeout_s) THEN
        Fault := TRUE;
        FaultId := 623; // Copley valid input telegram stale
    END_IF
ELSIF ResetRequest
      AND CommandIsZero
      AND NOT EncoderWcState
      AND NOT EncoderTxPdoState
      AND EncoderReady
      AND NOT EncoderError
      AND NOT CopleyWcState
      AND NOT Copley2WcState
      AND encoderToggleHealthy
      AND copleyToggleHealthy
      AND copley2ToggleHealthy THEN
    Fault := FALSE;
    FaultId := 0;
END_IF

SafeToDrive :=
    NOT Fault
    AND NOT EncoderWcState
    AND NOT EncoderTxPdoState
    AND EncoderReady
    AND NOT EncoderError
    AND NOT CopleyWcState
    AND NOT Copley2WcState
    AND encoderToggleHealthy
    AND copleyToggleHealthy
    AND copley2ToggleHealthy;

END_FUNCTION_BLOCK

// ---- POUs/FB_AllocationTransfer.TcPOU
FUNCTION_BLOCK FB_AllocationTransfer
VAR_INPUT
    Command : DUT_MotorDriverCommand;
    RuntimeRequestId : UDINT;
    CommissioningActive : BOOL;
    SourceControl : ARRAY [1..4] OF WORD;
    SourceTorque : ARRAY [1..4] OF INT;
    StatusWord : ARRAY [1..4] OF WORD;
    ActualCurrent : ARRAY [1..4] OF INT;
    PositionCount : DINT;
    VelocityCount : DINT;
    IoReady : BOOL;
    SourceFaultId : UDINT;
    Period100ns : UDINT;
END_VAR
VAR_OUTPUT
    Control : ARRAY [1..4] OF WORD;
    Torque : ARRAY [1..4] OF INT;
END_VAR
VAR
    i : INT;
    pairIndex : INT;
    idle : BOOL;
    servoEnabled : BOOL;
    weights : ARRAY [1..2] OF LREAL;
    weightedTorque : LREAL;
    cycleIndex : UDINT;
    sessionId : UDINT;
    sample : DUT_AllocationSample;
END_VAR

cycleIndex := cycleIndex + 1;
servoEnabled := (Command.ControlWord AND WORD#16#000F) = WORD#16#000F;
idle := NOT servoEnabled AND (Command.TargetTorque = 0)
    AND (ABS(VelocityCount) <= 1000) AND NOT CommissioningActive;
FOR i := 1 TO 4 DO
    idle := idle AND ((StatusWord[i] AND WORD#16#0004) = 0)
        AND (SourceTorque[i] = 0);
    Control[i] := SourceControl[i];
    Torque[i] := SourceTorque[i];
END_FOR

IF GVL_AllocationTransfer.RequestId <> GVL_AllocationTransfer.AckId THEN
    GVL_AllocationTransfer.RejectId := 0;
    IF NOT idle THEN
        GVL_AllocationTransfer.RejectId := 1; // no in-motion reconfiguration
    ELSIF NOT GVL_AllocationTransfer.RequestedEnabled THEN
        GVL_AllocationTransfer.Active := FALSE;
        GVL_AllocationTransfer.FaultId := 0;
    ELSE
        weights[1] := 1.0 + GVL_AllocationTransfer.RequestedBeta;
        weights[2] := 1.0 - GVL_AllocationTransfer.RequestedBeta * GVL_AllocationTransfer.RequestedRatio;
        pairIndex := UINT_TO_INT(GVL_AllocationTransfer.RequestedPair);
        IF NOT ((pairIndex >= 1) AND (pairIndex <= 3)
            AND ((pairIndex = 1) OR GVL_MotorRuntimeInternal.NORMAL_FOUR_AXIS_ENABLED)
            AND (GVL_AllocationTransfer.RequestedBeta >= -0.2)
            AND (GVL_AllocationTransfer.RequestedBeta <= 0.2)
            AND (GVL_AllocationTransfer.RequestedRatio >= 0.5)
            AND (GVL_AllocationTransfer.RequestedRatio <= 2.0)
            AND (weights[1] >= 0.8) AND (weights[1] <= 1.2)
            AND (weights[2] >= 0.8) AND (weights[2] <= 1.2)) THEN
            GVL_AllocationTransfer.RejectId := 2;
        ELSIF NOT IoReady OR (SourceFaultId <> 0) OR (Period100ns <> 2500) THEN
            GVL_AllocationTransfer.RejectId := 3;
        ELSIF (PositionCount < GVL_MotorRuntimeInternal.TORQUE_LINKAGE_LOWER_COUNT[pairIndex+1])
           OR (PositionCount > GVL_MotorRuntimeInternal.TORQUE_LINKAGE_UPPER_COUNT[pairIndex]) THEN
            GVL_AllocationTransfer.RejectId := 4;
        ELSE
            GVL_AllocationTransfer.Pair := GVL_AllocationTransfer.RequestedPair;
            GVL_AllocationTransfer.Beta := GVL_AllocationTransfer.RequestedBeta;
            GVL_AllocationTransfer.Ratio := GVL_AllocationTransfer.RequestedRatio;
            GVL_AllocationTransfer.Weights := weights;
            GVL_AllocationTransfer.Active := TRUE;
            GVL_AllocationTransfer.Started := FALSE;
            GVL_AllocationTransfer.Complete := FALSE;
            GVL_AllocationTransfer.FaultId := 0;
            sessionId := GVL_AllocationTransfer.RequestId;
        END_IF
    END_IF
    GVL_AllocationTransfer.AckId := GVL_AllocationTransfer.RequestId;
END_IF

IF GVL_AllocationTransfer.Active THEN
    IF servoEnabled AND NOT GVL_AllocationTransfer.Started THEN
        IF (RuntimeRequestId <> 0) AND (RuntimeRequestId = sessionId)
           AND NOT CommissioningActive THEN
            GVL_AllocationTransfer.Started := TRUE;
        ELSE
            // An abandoned arm must never change a later ordinary experiment.
            GVL_AllocationTransfer.Active := FALSE;
        END_IF
    END_IF
END_IF

IF GVL_AllocationTransfer.Active AND GVL_AllocationTransfer.Started THEN
    pairIndex := UINT_TO_INT(GVL_AllocationTransfer.Pair);
    IF CommissioningActive OR NOT IoReady OR (SourceFaultId <> 0)
       OR (Period100ns <> 2500)
       OR (servoEnabled AND (RuntimeRequestId <> sessionId))
       OR (PositionCount < GVL_MotorRuntimeInternal.TORQUE_LINKAGE_LOWER_COUNT[pairIndex+1])
       OR (PositionCount > GVL_MotorRuntimeInternal.TORQUE_LINKAGE_UPPER_COUNT[pairIndex]) THEN
        GVL_AllocationTransfer.FaultId := 630;
    END_IF
    FOR i := pairIndex TO pairIndex+1 DO
        weightedTorque := INT_TO_LREAL(SourceTorque[i]) * GVL_AllocationTransfer.Weights[i-pairIndex+1];
        // Physical scale is 0.1 A / 1000 counts. Abort instead of clipping
        // a trial whose changed allocation would exceed the existing 2 A.
        IF ABS(weightedTorque) > 20000.0 THEN
            GVL_AllocationTransfer.FaultId := 631;
        ELSE
            Torque[i] := LREAL_TO_INT(weightedTorque);
        END_IF
    END_FOR
END_IF

IF GVL_AllocationTransfer.FaultId <> 0 THEN
    FOR i := 1 TO 4 DO
        Control[i] := 0;
        Torque[i] := 0;
    END_FOR
END_IF

// Publish every cycle, including ordinary experiments and the final stop.
// The shared File Writer supplies the recording trigger and sample time.
sample.cycleIndex := cycleIndex;
sample.positionCount := PositionCount;
sample.velocityCount := VelocityCount;
sample.virtualTorque := INT_TO_DINT(Command.TargetTorque);
sample.faultId := SourceFaultId;
IF GVL_AllocationTransfer.FaultId <> 0 THEN sample.faultId := GVL_AllocationTransfer.FaultId; END_IF
sample.ioReady := BOOL_TO_DINT(IoReady);
sample.period100ns := Period100ns;
sample.requestId := 0;
IF GVL_AllocationTransfer.Active AND GVL_AllocationTransfer.Started THEN
    sample.requestId := sessionId;
END_IF
FOR i := 1 TO 4 DO
    sample.targetCurrent[i] := INT_TO_DINT(Torque[i]);
    IF NOT IoReady THEN sample.targetCurrent[i] := 0; END_IF
    sample.actualCurrent[i] := INT_TO_DINT(ActualCurrent[i]);
    sample.statusWord[i] := WORD_TO_DINT(StatusWord[i]);
END_FOR
GVL_AllocationTransfer.Snapshot := sample;

IF GVL_AllocationTransfer.Active AND GVL_AllocationTransfer.Started THEN
    IF NOT servoEnabled OR (GVL_AllocationTransfer.FaultId <> 0) THEN
        // One configuration covers exactly one servo-on interval. The next
        // experiment cannot silently inherit this trial's allocation.
        GVL_AllocationTransfer.Complete := TRUE;
        GVL_AllocationTransfer.Active := FALSE;
    END_IF
END_IF

END_FUNCTION_BLOCK
